// TIA Portal V17 export
// export: Created 2021-12-03T08:08:08.09202Z, ExportSetting WithDefaults, DisplayName Totally Integrated Automation Portal, DisplayVersion V17, DisplayName TIA Portal Openness, DisplayVersion V17, DisplayName TIA Portal Version Control Interface, DisplayVersion V17, DisplayName STEP 7 Professional, DisplayVersion V17, DisplayName STEP 7 Safety, DisplayVersion V17, DisplayName WinCC Advanced, DisplayVersion V17
VAR_GLOBAL   // PLC tag table "Data_Read"
   CmndON AT %MW400 : Word;   // Команды включения
   CmndON_0 AT %M400.0 : Bool;   // Команды включения
   CmndON_1 AT %M400.1 : Bool;   // Команды включения
   CmndON_2 AT %M400.2 : Bool;   // Команды включения
   CmndON_3 AT %M400.3 : Bool;   // Команды включения
   CmndON_4 AT %M400.4 : Bool;   // Команды включения
   CmndON_5 AT %M400.5 : Bool;   // Команды включения
   CmndON_6 AT %M400.6 : Bool;   // Команды включения
   CmndON_7 AT %M400.7 : Bool;   // Команды включения
   CmndON_8 AT %M401.0 : Bool;   // Команды включения
   CmndON_9 AT %M401.1 : Bool;   // Команды включения
   CmndON_10 AT %M401.2 : Bool;   // Команды включения
   CmndON_11 AT %M401.3 : Bool;   // Команды включения
   CmndON_12 AT %M401.4 : Bool;   // Команды включения
   CmndON_13 AT %M401.5 : Bool;   // Команды включения
   CmndON_14 AT %M401.6 : Bool;   // Команды включения
   CmndON_15 AT %M401.7 : Bool;   // Команды включения
   CmndOFF AT %MW404 : Word;   // Команды отключения
   CmndOFF_0 AT %M404.0 : Bool;   // Команды отключения
   CmndOFF_1 AT %M404.1 : Bool;   // Команды отключения
   CmndOFF_2 AT %M404.2 : Bool;   // Команды отключения
   CmndOFF_3 AT %M404.3 : Bool;   // Команды отключения
   CmndOFF_4 AT %M404.4 : Bool;   // Команды отключения
   CmndOFF_5 AT %M404.5 : Bool;   // Команды отключения
   CmndOFF_6 AT %M404.6 : Bool;   // Команды отключения
   CmndOFF_7 AT %M404.7 : Bool;   // Команды отключения
   CmndOFF_8 AT %M405.0 : Bool;   // Команды отключения
   CmndOFF_9 AT %M405.1 : Bool;   // Команды отключения
   CmndOFF_10 AT %M405.2 : Bool;   // Команды отключения
   CmndOFF_11 AT %M405.3 : Bool;   // Команды отключения
   CmndOFF_12 AT %M405.4 : Bool;   // Команды отключения
   CmndOFF_13 AT %M405.5 : Bool;   // Команды отключения
   CmndOFF_14 AT %M405.6 : Bool;   // Команды отключения
   CmndOFF_15 AT %M405.7 : Bool;   // Команды отключения
   Cmnd_AckRst AT %MW408 : Word;   // Команды сброса
   Cmnd_AckRst_0 AT %M408.0 : Bool;   // Команды сброса
   Cmnd_AckRst_1 AT %M408.1 : Bool;   // Команды сброса
   Cmnd_AckRst_2 AT %M408.2 : Bool;   // Команды сброса
   Cmnd_AckRst_3 AT %M408.3 : Bool;   // Команды сброса
   Cmnd_AckRst_4 AT %M408.4 : Bool;   // Команды сброса
   Cmnd_AckRst_5 AT %M408.5 : Bool;   // Команды сброса
   Cmnd_AckRst_6 AT %M408.6 : Bool;   // Команды сброса
   Cmnd_AckRst_7 AT %M408.7 : Bool;   // Команды сброса
   Cmnd_AckRst_8 AT %M409.0 : Bool;   // Команды сброса
   Cmnd_AckRst_9 AT %M409.1 : Bool;   // Команды сброса
   Cmnd_AckRst_10 AT %M409.2 : Bool;   // Команды сброса
   Cmnd_AckRst_11 AT %M409.3 : Bool;   // Команды сброса
   Cmnd_AckRst_12 AT %M409.4 : Bool;   // Команды сброса
   Cmnd_AckRst_13 AT %M409.5 : Bool;   // Команды сброса
   Cmnd_AckRst_14 AT %M409.6 : Bool;   // Команды сброса
   Cmnd_AckRst_15 AT %M409.7 : Bool;   // Команды сброса
   CmndSwitch AT %MW410 : Word;   // Команды переключения
   CmndSwitch_0 AT %M410.0 : Bool;   // Команды переключения
   CmndSwitch_1 AT %M410.1 : Bool;   // Команды переключения
   CmndSwitch_2 AT %M410.2 : Bool;   // Команды переключения
   CmndSwitch_3 AT %M410.3 : Bool;   // Команды переключения
   CmndSwitch_4 AT %M410.4 : Bool;   // Команды переключения
   CmndSwitch_5 AT %M410.5 : Bool;   // Команды переключения
   CmndSwitch_6 AT %M410.6 : Bool;   // Команды переключения
   CmndSwitch_7 AT %M410.7 : Bool;   // Команды переключения
   CmndSwitch_8 AT %M411.0 : Bool;   // Команды переключения
   CmndSwitch_9 AT %M411.1 : Bool;   // Команды переключения
   CmndSwitch_10 AT %M411.2 : Bool;   // Команды переключения
   CmndSwitch_11 AT %M411.3 : Bool;   // Команды переключения
   CmndSwitch_12 AT %M411.4 : Bool;   // Команды переключения
   CmndSwitch_13 AT %M411.5 : Bool;   // Команды переключения
   CmndSwitch_14 AT %M411.6 : Bool;   // Команды переключения
   CmndSwitch_15 AT %M411.7 : Bool;   // Команды переключения
   Service_Button1 AT %MW412 : Word;   // Кнопки в сервисном меню
   Service_Button1_0 AT %M412.0 : Bool;   // Кнопки в сервисном меню
   Service_Button1_1 AT %M412.1 : Bool;   // Кнопки в сервисном меню
   Service_Button1_2 AT %M412.2 : Bool;   // Кнопки в сервисном меню
   Service_Button1_3 AT %M412.3 : Bool;   // Кнопки в сервисном меню
   Service_Button1_4 AT %M412.4 : Bool;   // Кнопки в сервисном меню
   Service_Button1_5 AT %M412.5 : Bool;   // Кнопки в сервисном меню
   Service_Button1_6 AT %M412.6 : Bool;   // Кнопки в сервисном меню
   Service_Button1_7 AT %M412.7 : Bool;   // Кнопки в сервисном меню
   Service_Button1_8 AT %M413.0 : Bool;   // Кнопки в сервисном меню
   Service_Button1_9 AT %M413.1 : Bool;   // Кнопки в сервисном меню
   Service_Button1_10 AT %M413.2 : Bool;   // Кнопки в сервисном меню
   Service_Button1_11 AT %M413.3 : Bool;   // Кнопки в сервисном меню
   Service_Button1_12 AT %M413.4 : Bool;   // Кнопки в сервисном меню
   Service_Button1_13 AT %M413.5 : Bool;   // Кнопки в сервисном меню
   Service_Button1_14 AT %M413.6 : Bool;   // Кнопки в сервисном меню
   Service_Button1_15 AT %M413.7 : Bool;   // Кнопки в сервисном меню
   Service_Button2 AT %MW414 : Word;   // Кнопки в сервисном меню
   Service_Button2_0 AT %M414.0 : Bool;   // Кнопки в сервисном меню
   Service_Button2_1 AT %M414.1 : Bool;   // Кнопки в сервисном меню
   Service_Button2_2 AT %M414.2 : Bool;   // Кнопки в сервисном меню
   Service_Button2_3 AT %M414.3 : Bool;   // Кнопки в сервисном меню
   Service_Button2_4 AT %M414.4 : Bool;   // Кнопки в сервисном меню
   Service_Button2_5 AT %M414.5 : Bool;   // Кнопки в сервисном меню
   Service_Button2_6 AT %M414.6 : Bool;   // Кнопки в сервисном меню
   Service_Button2_7 AT %M414.7 : Bool;   // Кнопки в сервисном меню
   Service_Button2_8 AT %M415.0 : Bool;   // Кнопки в сервисном меню
   Service_Button2_9 AT %M415.1 : Bool;   // Кнопки в сервисном меню
   Service_Button2_10 AT %M415.2 : Bool;   // Кнопки в сервисном меню
   Service_Button2_11 AT %M415.3 : Bool;   // Кнопки в сервисном меню
   Service_Button2_12 AT %M415.4 : Bool;   // Кнопки в сервисном меню
   Service_Button2_13 AT %M415.5 : Bool;   // Кнопки в сервисном меню
   Service_Button2_14 AT %M415.6 : Bool;   // Кнопки в сервисном меню
   Service_Button2_15 AT %M415.7 : Bool;   // Кнопки в сервисном меню
END_VAR
